(* PLC project Unnamed, Unknown Unnamed 1 *)
(* stored: creationDateTime 2020-01-27T09:18:59, modificationDateTime 2020-08-02T12:59:54 *)

PROGRAM program0
  VAR
    TIMER : TIME := T#4s;
    TE : TIME := T#0s;
    reset : BOOL;
  END_VAR
  VAR
    V_Pump AT %QX0.0 : BOOL;
    Lid AT %QX0.1 : BOOL;
    Vent AT %QX0.2 : BOOL;
    Bar AT %QX0.3 : BOOL;
    Seal1 AT %QX0.4 : BOOL;
    Seal2 AT %QX0.5 : BOOL;
    Pump_Start AT %IX0.2 : BOOL;
    Pump_stop AT %IX0.3 : BOOL;
    START_CYCLE AT %IX0.4 : BOOL;
  END_VAR
  VAR
    FINISH_CYCLE : BOOL;
    hold1I : BOOL;
    TOF0 : TOF;
    TOF1 : TOF;
    TOF2 : TOF;
    R_TRIG0 : R_TRIG;
    R_TRIG1 : R_TRIG;
  END_VAR
  VAR  (* added by the conversion: wires and edge detectors of the diagram *)
    F_TRIG1 : F_TRIG;
  END_VAR

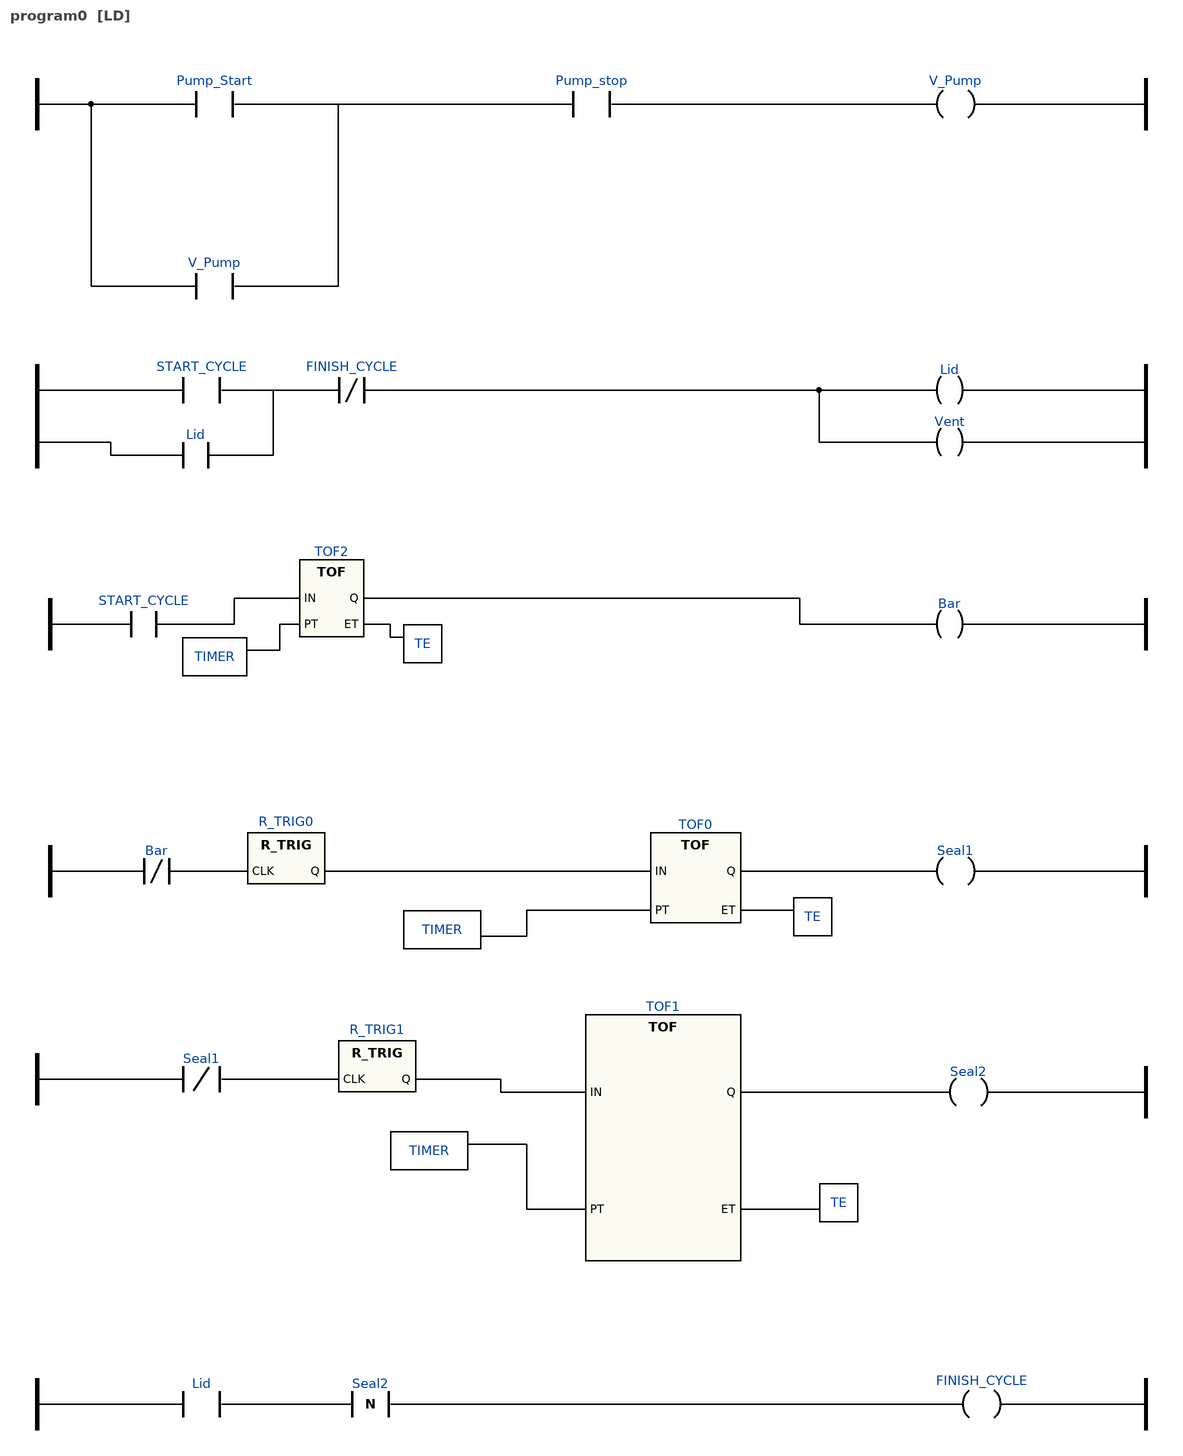
(* LD diagram, written out as Structured Text *)
V_Pump := (Pump_Start OR V_Pump) AND Pump_stop;
Lid := (START_CYCLE OR Lid) AND NOT FINISH_CYCLE;
Vent := (START_CYCLE OR Lid) AND NOT FINISH_CYCLE;
TOF2(IN := START_CYCLE, PT := TIMER);
Bar := TOF2.Q;
TE := TOF2.ET;
R_TRIG0(CLK := NOT Bar);
TOF0(IN := R_TRIG0.Q, PT := TIMER);
Seal1 := TOF0.Q;
TE := TOF0.ET;
R_TRIG1(CLK := NOT Seal1);
TOF1(IN := R_TRIG1.Q, PT := TIMER);
Seal2 := TOF1.Q;
TE := TOF1.ET;
F_TRIG1(CLK := Seal2);
FINISH_CYCLE := Lid AND F_TRIG1.Q;
END_PROGRAM

FUNCTION_BLOCK TP_WITH_RESET
  VAR_INPUT
    IN : BOOL;
    PT : TIME := T#4s;
    RESET : BOOL;
  END_VAR
  VAR_OUTPUT
    Q : BOOL;
    ET : TIME := T#0s;
  END_VAR
  VAR
    STATE : SINT := 0;
    PREV_IN : BOOL := FALSE;
    CURRENT_TIME : TIME;
    START_TIME : TIME;
  END_VAR

            (* Pragma to set current time *)
{__SET_VAR(data__->,CURRENT_TIME,,__CURRENT_TIME)}

(*Timer block code *)
IF ((STATE = 0) AND NOT(PREV_IN) AND IN) THEN  (* found rising edge on IN *)
    (* start timer... *)
    STATE := 1;
    Q := TRUE;
    START_TIME := CURRENT_TIME;

ELSIF (STATE = 1) THEN (* timer counting *)
    IF ((START_TIME + PT) <= CURRENT_TIME) THEN (* timer expired *)
        STATE := 2;
        Q := FALSE;
        ET := PT;
    ELSE (* continue counting *)
        ET := CURRENT_TIME - START_TIME;
    END_IF;
END_IF;

IF ((STATE = 2) AND NOT(IN)) THEN
    ET := T#0s;
    STATE := 0;
END_IF;

IF (RESET) THEN (* reset pressed *)
  ET := T#0s;
  STATE := 0;
  Q := FALSE;
END_IF;

PREV_IN := IN;
          
END_FUNCTION_BLOCK

CONFIGURATION Config0
  RESOURCE Res0 ON PLC
    TASK task0(INTERVAL := T#20ms, PRIORITY := 0);
    PROGRAM instance0 WITH task0 : program0;
  END_RESOURCE
END_CONFIGURATION
